// TIA Portal V17 export
// export: Created 2025-06-26T06:49:32.6031032Z, ExportSetting WithDefaults, DisplayName Totally Integrated Automation Portal, DisplayVersion V17 Update 8, DisplayName TIA Portal Openness, DisplayVersion V17 Update 8, DisplayName TIA Portal Version Control Interface, DisplayVersion V17, DisplayName STEP 7 Professional, DisplayVersion V17 Update 8, DisplayName STEP 7 Safety, DisplayVersion V17 Update 6, DisplayName WinCC Advanced, DisplayVersion V17 Update 8
TYPE "CurrentSetting-STRUCT"
// stored: IsFailsafeCompliant false
   STRUCT
      Fluid { S7_SetPoint := 'True'} : "FluidData-STRUCT";   // Kältemittelspezifische Einstellungen (Wird aus StaticData entnommen)
      Compressor { S7_SetPoint := 'True'} : "CompressorData-STRUCT";   // Kompressorspezifische Einstellungen (Wird aus StaticData entnommen)
      System { S7_SetPoint := 'True'} : "SystemData-STRUCT";   // Systemspezifische Einstellungen (Wird aus StaticData entnommen)
      VariableSetting { S7_SetPoint := 'True'} : "VariableSetting-STRUCT";   // Einstellungen, die über die HMI voreingestellt werden können
      StaticSetting { S7_SetPoint := 'True'} : "StaticSetting-STRUCT";   // Programmparameter um Systemverhalten Abzustimmen
      NewInitialisation_Required : Bool;   // Gets set on configuration changes and reset on restart
      ParameterSet_Ordered : Bool;   // Shows if the parameterset is successfully loaded
      ParameterSet_Indicator : Bool;
      MissingSetting : Struct   // Catch all category. To be sorted.
         Compressor : Struct
            OilPumpCurveCritical : Real := 0.133;   // [kPa/rpm] Minimum adequate oil pump performance
            OilPumpCurveWarning : Real := 0.166;   // [kPa/rpm] Minimum expected oil pump performance
            MinStartupSpeed : Real := 25.0;   // [rpm] Minimum speed at compressor start
            WarmupSpeed : Real := 550.0;   // [rpm] Speed in warmup state
            MinOperationalSpeed : Real := 550.0;   // [rpm] Minimum speed in operation
            MaxOperationalSpeed : Real := 1200.0;   // [rpm] Maximum speed in operation
            OilFilterDeltaPCritical : Real := 150.0;   // [kPa] Maximum oil filter delta P
            OilFilterDeltaPWarning : Real := 100.0;   // [kPa] Warning oil filter delta P
         END_STRUCT;
         System : Struct
            HydrolockSpeed : Real := 330.0;   // [rpm] Max safe speed under hydrolock conditions
            CondenserCoefficient : Real := 13.024;   // [?] Mass flow calculation
            EvaporatorCoefficient : Real := 19.07;   // [?] Mass flow calculation
            SuctionLineDryLimitPressure : Real := 80.0;   // [kPa] Compressor suction pressue when suction line is considered dry
            SuctionLineDryLimitSuperheat : Real := 27.0;   // [C] Compressor suction superheat when suction line is considered dry
            CompressorSuperheatDischargeMinimum : Real := 20.0;   // [C] Lowest permissible compressor discharge superheat in operation
            RecuperatorDeltaTWorking : Real := 3.0;   // [C] Recuperator superheat gain when it is considered working
            RecuperatorDeltaTNotWorking : Real := -2.0;   // [C] Recuperator superheat gain when it is considered not working (can be negative)
            ExpansionValvePositionStart : Real := 5.5;   // [%] Expansion valve position in State 4 Start
            ExpansionValvePositionStartCold : Real := 3.0;   // [%] Expansion valve position in State 4 Start, cold start
            HeatSourceDeltaPFlow : Real := 2.0;   // [kPa] Delta P over the heat source that indicates flow
            HeatSinkDeltaPFlow : Real := 2.0;   // [kPa] Delta P over the heat sink that indicates flow
         END_STRUCT;
         Misc : Struct   // A lot of odds and ends
            CompressorStoppedLimit : Real := 10.0;   // [rpm] Compressor speed at which it is considered stopped
            State2DwellTime { S7_SetPoint := 'True'} : Time := T#10s;   // Standby
            State3DwellTime : Time := T#30s;   // Prepare start
            State4DwellTime : Time := T#30s;   // Start
            State5DwellTime : Time := T#20m;   // Warmup
            State7DwellTime : Time := T#10s;   // Stop
            State2PauseTime : Time := T#10s;   // Minimum pause in standby before resume
            EmergencyStopWaitTime : Time := T#5m;   // Cooldown pause after Emergency stop is reset
            T_HeatSinkTemperatureIn_Max : Real := 75.0;   // [C] Maximum temperature on the suction side of the heat sink
         END_STRUCT;
      END_STRUCT;
   END_STRUCT;
END_TYPE
